FUNCTION_BLOCK FB_TcLogger IMPLEMENTS I_Logger
VAR_INPUT
	eLogLevel:					E_Event;
END_VAR
VAR_OUTPUT
END_VAR
VAR_IN_OUT

END_VAR
VAR
END_VAR

METHOD M_Log
VAR_INPUT
	stEvent	: 		ST_Event;
END_VAR

VAR
	sMessage:			STRING(255);
END_VAR
////IF stEvent.New THEN
//	sMessage:= Concat(Concat(stEvent.Instance, ' | '), stEvent.Message);
//	CASE stEvent.EventType OF
//		E_Event.Error:
//			ADSLOGSTR( msgCtrlMask := ADSLOG_MSGTYPE_ERROR , msgFmtStr := sMessage, strArg := '');
//		E_Event.Warning:
//			ADSLOGSTR( msgCtrlMask := ADSLOG_MSGTYPE_WARN , msgFmtStr := sMessage, strArg := '');
//		E_Event.Information:
//			ADSLOGSTR( msgCtrlMask := ADSLOG_MSGTYPE_HINT , msgFmtStr := sMessage, strArg := '');
//		E_Event.Debug:
//			ADSLOGSTR( msgCtrlMask := ADSLOG_MSGTYPE_HINT, msgFmtStr := sMessage, strArg := '');
//		E_Event.Verbose:
//			ADSLOGSTR( msgCtrlMask := ADSLOG_MSGTYPE_HINT , msgFmtStr := sMessage, strArg := '');
//	END_CASE
////END_IF
END_METHOD

END_FUNCTION_BLOCK

(* stored: Version 1.1.0.1, ProductVersion 3.1.4024.12
   POU FB_TcLogger: Id {f9ae1251-8db7-0f83-3fe4-63ffe332e5de}, SpecialFunc None
   Method M_Log: Id {559b0423-33fe-0a3c-0dca-60935fba72a8} *)
